TYPE SampleTaskFunctionBuffer :
STRUCT
	x : LREAL;
	y : LREAL;
END_STRUCT
END_TYPE

(* stored: Version 1.1.0.1, ProductVersion 3.1.4024.9
   DUT SampleTaskFunctionBuffer: Id {53505139-cecc-02de-0b16-cae034b45e5a} *)
